TYPE "UDT_HMI_Alarm_V2"
VERSION : 0.1
   STRUCT
      t : Struct
         x0 : Bool;
         x1 : Bool;
         x2 : Bool;
         x3 : Bool;
         x4 : Bool;
         x5 : Bool;
         x6 : Bool;
         x7 : Bool;
         x8 : Bool;
         x9 : Bool;
         x10 : Bool;
         x11 : Bool;
         x12 : Bool;
         x13 : Bool;
         x14 : Bool;
         x15 : Bool;
      END_STRUCT;
      iHmiSumAlm : Word;
   END_STRUCT;

END_TYPE

TYPE "UDT_SelvMa_Allarm"
VERSION : 0.1
   STRUCT
      tEmergencyAlarm { ExternalWritable := 'False'} : Array["STARTARRAY".."DALARM"] of "UDT_HMI_Alarm_V2";
      tAlarm { ExternalWritable := 'False'} : Array["STARTARRAY".."DALARM"] of "UDT_HMI_Alarm_V2";
      tWarning { ExternalWritable := 'False'} : Array["STARTARRAY".."DALARM"] of "UDT_HMI_Alarm_V2";
   END_STRUCT;

END_TYPE

DATA_BLOCK "SelvMaFrame_Hmi"
{ S7_Optimized_Access := 'FALSE' }
VERSION : 0.1
   STRUCT
      tFr : Array["STARTARRAY".."DNUMFRAME"] of Struct
         tHMR : Struct   // {[Unit]|[Scada Unit]|[LowLimit]|[HigLimit]|[Acces]}
            xFrameEnabled : Bool;   // Enabled - Frame {x|x|x|x|O}
            xMaintenanceModeEnabled : Bool;   // Maintenance Mode Enable {x|x|x|x|O}
            xManualCommandEnabled : Bool;   // Manual Mode Enable {x|x|x|x|O}
            dActualPosition_cmm : DInt;   // Actual Position {cmm|cmm|x|x|O}
            rActualPosition_mm : Real;   // Actual Position {mm|mm|x|x|O}
            dTarget_cmm : DInt;   // Target Section  {cmm|mm|x|x|O}
            rTarget_mm : Real;   // Target Section  {mm|mm|x|x|O}
            dFinalTarget_cmm : DInt;   // Final Target Section  {cmm|mm|x|x|O}
            rFinalTarget_mm : Real;   // Final Target Section  {mm|mm|x|x|O}
            dOffsetSingleSection_cmm : DInt;   // Offset single Target Section  {cmm|mm|x|x|O}
            rOffsetSingleSection_mm : Real;   // Offset single Target Section  {mm|mm|x|x|O}
            dOffseTotalSection_cmm : DInt;   // Offset Total Section  {cmm|mm|x|x|O}
            rOffseTotalSection_cmm : Real;   // Offset Total Section {mm|mm|x|x|O}
            iState : Int;   // Machine State (1=Ready, 3=Run, 7=Anomaly) {x|x|x|x|O}
            tManCmd : Struct
               xForwardTraslation : Bool;   // Forward traslation {x|x|x|x|O}
               xBackwardTraslation : Bool;   // Backward traslation {x|x|x|x|O}
               xPositioningCmd : Bool;
            END_STRUCT;
         END_STRUCT;
         tHMW : Struct   // {[Unit]|[Scada Unit]|[LowLimit]|[HigLimit]|[Acces]}
            xEnableFrame : Bool;   // Enabled - Frame  {x|x|x|x|O}
            xDisableFrame : Bool;   // Disabled - Frame  {x|x|x|x|O}
            xEnableDisableManualCommand : Bool;   // Enable Disable Manual Command {x|x|x|x|O}
            xPresetEncoder : Bool;   // Preset Encoder  {x|x|x|x|O}
            xEnDisMaintenance : Bool;   // Enable disable Maintenance service
            dPositionManCmd_cmm : DInt;   // Positioning Manual Cmd  {cmm|cmm|x|x|O}
            rPositionManCmd_mm : Real;   // Positioning Manual Cmd  {mm|mm|x|x|O}
            tManCmd : Struct
               xForwardTraslation : Bool;   // Forward traslation {x|x|x|x|O}
               xBackwardTraslation : Bool;   // Backward traslation {x|x|x|x|O}
               xPositioningCmd : Bool;
            END_STRUCT;
         END_STRUCT;
      END_STRUCT;
   END_STRUCT;


BEGIN

END_DATA_BLOCK

DATA_BLOCK "SelvMaFrame_Alm"
{ S7_Optimized_Access := 'FALSE' }
VERSION : 0.1
NON_RETAIN
   STRUCT
      Fr : Array["STARTARRAY".."DNUMFRAME"] of "UDT_SelvMa_Allarm";
   END_STRUCT;


BEGIN

END_DATA_BLOCK

